(* IEC 61131-3 sources: Guziczki_i_swiatelka/Guziczki_i_swiatelka/Temp/History/18/Program1, 1 file *)

(* ---- Cyclic.st ---- *)
PROGRAM _CYCLIC
	PWM_1(duty_cycle :=30, period :=T#1s , input_PWM :=input_3 );
IF PWM_1.out THEN
	output_5 := TRUE;
	output_6 := TRUE;
	END_IF;

END_PROGRAM
